Fanuc KAREL source: SET_JPOS_REG.kl

PROGRAM T
%NOLOCKGROUP
VAR
 v0 : INTEGER
 v1 : JOINTPOS
 v2 : INTEGER
 v3 : INTEGER
BEGIN
 SET_JPOS_REG(v0, v1, v2, v3)
END T
